Staubli VAL3: onEnterEvent.pgx

program onEnterEvent()
  local num i
  local num l_nIndex
  local string l_sItem[2]
  local num l_nResult
  local string l_sMessage
begin
  //
  // NB sEvent is the selected
  // element in the LIST
  //
  if sEvent!=""
    logMsg("Page trajectory trajtype "+trajType:libPath())
    //
    l_sItem=sEvent
    call trajType:onEdit(l_sItem)
    if find(l_sItem,"Disk://")!=-1 and l_nResult==0
      // load the page
      call loadPage(l_sItem,l_sItem[1])
    endIf
    // logMsg
    logMsg("[KERNEL] INTERFACE:PAGE Edit trajectory")
    //
    call buildList()
  endIf
  //
end
